TYPE ST_PNController_Set :
STRUCT

END_STRUCT
END_TYPE

(* stored: Version 1.1.0.1, ProductVersion 3.1.4024.12
   DUT ST_PNController_Set: Id {9d99ae19-2b04-4caf-b3af-7cc0aa67da30} *)
